// TwinCAT 3 PLC project CoE_Read_Write
// ProgramVersion: 3.1.4024.0
// libraries:
//   Tc2_EtherCAT, * (Beckhoff Automation GmbH)
//   Tc2_Standard, * (Beckhoff Automation GmbH)
//   Tc2_System, * (Beckhoff Automation GmbH)
//   Tc3_Module, * (Beckhoff Automation GmbH)
//   VisuDialogs, * (System)
// project tree:
//   / GlobalTextList.TcGTLO, PlcTask.TcTTO, Visualization Manager.TcVMO (not stored)
//   POUs/ fbEcCoESdoRead.TcPOU, FB_EcCoESdoWrite.TcPOU, MAIN.TcPOU, Read_Write_CoE.TcPOU, Test_FB.TcPOU
//   VISUs/ V002_CB_Config.TcVIS
// real-time tasks:
//   TASK PlcTask: cycle T#10ms, priority 20, ADS port 350
// I/O:
//   DEVICE Device 2 (EtherCAT), AmsNetId 169.254.127.131.3.1
//     Term 1 (EK1100) [EK1100 EtherCAT Coupler (2A E-Bus)]
//       Term 2 (EL5072) [EL5072 2Ch. Inductive sensor interface (LVDT, Half Bridge)]
//       Term 3 (EL9011) [EL9011 End Terminal]
// variable links:
//   CoE_Read_Write/CoE_Read_Write Instance <-> Device 2 (EtherCAT)/Term 1 (EK1100)/Term 2 (EL5072)
//     PlcTask Inputs/Read_Write_CoE.SlaveNetID <-> InfoData/AdsAddr/netId
//     PlcTask Inputs/Read_Write_CoE.SlavePort <-> InfoData/AdsAddr/port

CONFIGURATION CoE_Read_Write
    RESOURCE PLC ON TwinCAT3
        TASK PlcTask(INTERVAL := T#10ms, PRIORITY := 20);
        PROGRAM MAIN WITH PlcTask : MAIN;
    END_RESOURCE
END_CONFIGURATION

// ---- POUs/MAIN.TcPOU

PROGRAM MAIN
VAR

END_VAR

Read_Write_CoE();

END_PROGRAM

// ---- POUs/Read_Write_CoE.TcPOU
PROGRAM Read_Write_CoE
VAR
	fbEcCoESdoRead			: FB_EcCoESdoRead;
	bReadSensitivity1  : BOOL;
	FB_EcCoESdoWriteEx		: FB_EcCoESdoWriteEx;
	bWriteSensitivity1 : BOOL;
 	SlaveNetID 	AT %I* 	    : T_AmsNetIdArr;			(* AMS Net ID *)
	SlavePort  	AT %I*  	    : WORD;				(* Port number *)
    nIndex          : WORD; (* CANopen Sdo index.*)
	
	fSensitivity_Live		    : REAL; 				(* Analog Input Limit 1 *)
	fSensitivity_ToUpload		    : REAL; 				(* Analog Input Limit 1 *)

	bReadError      : BOOL;
        nReadErrId      : UDINT;
	bWriteError     : BOOL;
        nWriteErrId     : UDINT;
	tTimeout         : TIME := DEFAULT_ADS_TIMEOUT;
	fSensitivity1: INT;	

	Upload: BOOL := TRUE;
END_VAR


(* Read the Analog Input Limit 1 CoE parameter *)
fbEcCoESdoRead(
	sNetId:= F_CreateAmsNetId(SlaveNetID), 
	nSlaveAddr:= SlavePort, 
	nSubIndex:= 16#16, (* Subindex of CoE Object *)
	nIndex:= 16#8001 , (* CoE Object Index *)
	pDstBuf:= ADR(fSensitivity_Live), 
	cbBufLen:= SIZEOF(fSensitivity_Live), 
	bExecute:= bReadSensitivity1, 
	tTimeout:= tTimeout, 
	bBusy=> , 
	bError=> bReadError, 
	nErrId=> nReadErrId, 
	cbRead=> );
	
	
(* Write to Analog Input Limit 1 CoE parameter *)
FB_EcCoESdoWriteEx(
	sNetId:= F_CreateAmsNetId(SlaveNetID), 
	nSlaveAddr:=SlavePort ,
	nSubIndex:=16#16, (* Subindex of CoE Object *)
	nIndex:=16#8001 , (* CoE Object Index *)
	pSrcBuf:=ADR(fSensitivity_ToUpload) ,
	cbBufLen:=SIZEOF(fSensitivity_ToUpload) ,
	bExecute:= bWriteSensitivity1,(* TRUE activate writing *)
	tTimeout:= tTimeout,
	bBusy=> ,
	bError=> ,
	nErrId=> );

	IF NOT FB_EcCoESdoWriteEx.bBusy THEN
		bWriteSensitivity1 := FALSE;
		IF NOT FB_EcCoESdoWriteEx.bError THEN
			(* write successful *)
			bWriteError := FALSE;
			nWriteErrId := 0;
		ELSE
			(* write failed *)
			bWriteError := FB_EcCoESdoWriteEx.bError;
			nWriteErrId := FB_EcCoESdoWriteEx.nErrId;
		END_IF
		FB_EcCoESdoWriteEx(bExecute := FALSE);
	END_IF

END_PROGRAM

// ---- POUs/fbEcCoESdoRead.TcPOU
FUNCTION_BLOCK fbEcCoESdoRead
VAR_INPUT
END_VAR
VAR_OUTPUT
END_VAR
VAR

	FB_EcCoESdoRead: FB_EcCoESdoRead;
END_VAR

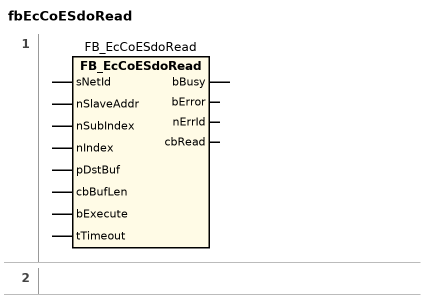
// NETWORK 1
FB_EcCoESdoRead();

// NETWORK 2

END_FUNCTION_BLOCK

// ---- POUs/FB_EcCoESdoWrite.TcPOU
FUNCTION_BLOCK FB_EcCoESdoWrite
VAR_INPUT
END_VAR
VAR_OUTPUT
END_VAR
VAR
FB_EcCoESdoWriteEx : FB_EcCoESdoWriteEx;

END_VAR

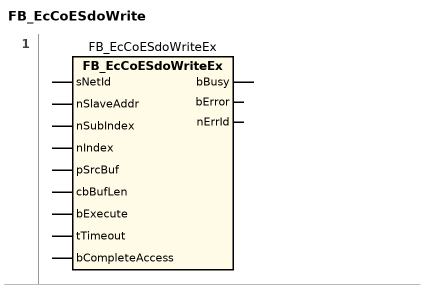
// NETWORK 1
FB_EcCoESdoWriteEx();

END_FUNCTION_BLOCK

// ---- POUs/Test_FB.TcPOU
FUNCTION_BLOCK Test_FB

VAR
nCounter	:	LINT;	
END_VAR

nCounter := nCounter + 1;

END_FUNCTION_BLOCK

// ---- GlobalTextList.TcGTLO
TEXTLIST GlobalTextList
  605 = '%0.2f'
  570 = '%0.6f'
  3131 = '>'
  21 = 'Gain'
  1375 = 'LVDT - Depth'
  1626 = 'Read Values'
  1977 = 'Sensitivity (mV/V/mm)'
  322 = 't##'
  871 = 'Write New'
END_TEXTLIST

// ---- VISUs/V002_CB_Config.TcVIS
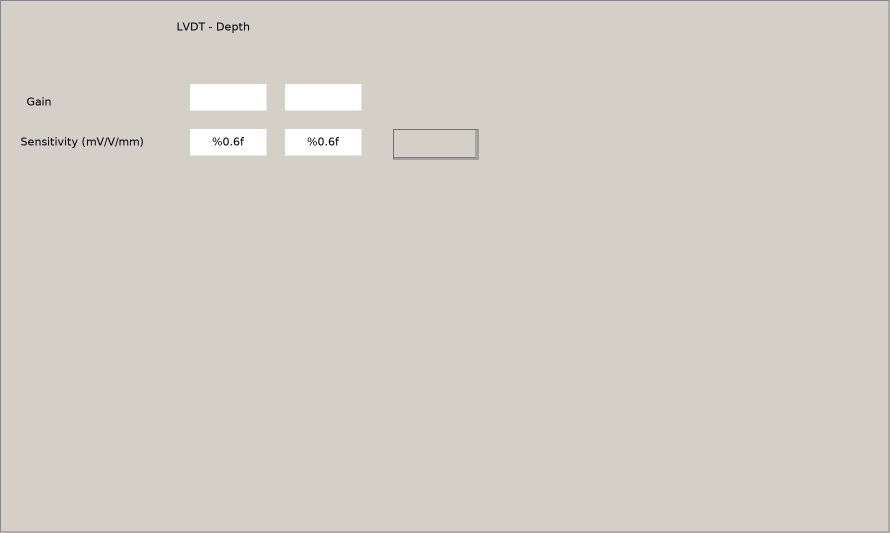
VISUALIZATION V002_CB_Config  // 890x533
    Textfield (284,83 78x28)
    Label (139,12 149x30), "LVDT - Depth"
    Label (11,87 56x30), "Gain"
    Label (15,127 135x30), "Sensitivity (mV/V/mm)"
    Textfield (284,128 78x28), "%0.6f", text variable: Read_Write_CoE.fSensitivity_ToUpload
        OnMouseClick: write Read_Write_CoE.fSensitivity_ToUpload via VisuDialogs.Numpad
    Textfield (189,83 78x28)
    Textfield (189,128 78x28), "%0.6f", text variable: Read_Write_CoE.fSensitivity_Live, input disabled if: TRUE
    Button (393,129 85x30)
        OnMouseDown: toggle Read_Write_CoE.bWriteSensitivity1
        OnMouseUp: toggle Read_Write_CoE.bReadSensitivity1
END_VISUALIZATION
